// TIA Portal V20 export
DATA_BLOCK "DB_SystemSSR"   // DB5
// stored: Access Published, MemoryReserve 100, Namespace Global
   VAR
      FromHMI : Struct
         Line : Struct
            A1 : "Global.SystemSSR";
            B1 { S7_SetPoint := 'True'} : "Global.SystemSSR";
            C1 { S7_SetPoint := 'True'} : "Global.SystemSSR";
            D1 { S7_SetPoint := 'True'} : "Global.SystemSSR";
         END_STRUCT;
      END_STRUCT;
      Line : Struct
         A1 : "Global.SystemSSR";
         B1 { S7_SetPoint := 'True'} : "Global.SystemSSR";
         C1 { S7_SetPoint := 'True'} : "Global.SystemSSR";
         D1 { S7_SetPoint := 'True'} : "Global.SystemSSR";
      END_STRUCT;
   END_VAR
BEGIN
END_DATA_BLOCK
